// TIA Portal V19 export
TYPE "LEXCHANGETRAY_typeHandlingXyzEm_toConstraintRollerDeliver"
// stored: Access Published
   STRUCT
      feedback : "LEXCHANGETRAY_typeHandlingXyzEm_toConstraintRollerFeedback";
      req : "LEXCHANGETRAY_typeHandlingXyzEm_toConstraintRollerReq";
   END_STRUCT;
END_TYPE
